{attribute 'linkalways'} 
{attribute 'no_explicit_call' := 'This FB is a CLASS and must be accessed using methods or properties'}
{attribute 'enable_dynamic_creation'}
FUNCTION_BLOCK _ETcVnContoursMatchComparisonMethod EXTENDS EnumDatatypeBase
VAR
	localData : ETcVnContoursMatchComparisonMethod;
	activeData : REFERENCE TO ETcVnContoursMatchComparisonMethod;
	enumBaseDatatype : _DINT(localData);
END_VAR

METHOD PRIVATE AddLocalEnumeration
VAR_INPUT
	Enumeration : T_MAXSTRING;
	Value : ETcVnContoursMatchComparisonMethod;
END_VAR
AddEnumeration(Enumeration, Value);
END_METHOD

PROPERTY PUBLIC Address : PVOID
GET
Address := ADR(activeData);
END_GET
END_PROPERTY

METHOD PUBLIC ClearReference
VAR_INPUT
END_VAR
activeData REF= localData;
SetBaseDatatypeReference();
END_METHOD

METHOD PUBLIC Clone : I_Datatype
VAR
    pClone : POINTER TO _ETcVnContoursMatchComparisonMethod;
END_VAR
pClone := __NEW(_ETcVnContoursMatchComparisonMethod(InitialValue := Value));
Clone := pClone^;
END_METHOD

METHOD FB_init : BOOL
VAR_INPUT
	bInitRetains : BOOL; // if TRUE, the retain variables are initialized (warm start / cold start)
	bInCopyCode : BOOL;  // if TRUE, the instance afterwards gets moved into the copy code (online change)
	InitialValue : ETcVnContoursMatchComparisonMethod;
END_VAR
localData := InitialValue;
AddBaseDatatype(enumBaseDatatype);
ClearReference();

AddLocalEnumeration('TCVN_CMCM_CONTOURS_MATCH_I1', ETcVnContoursMatchComparisonMethod.TCVN_CMCM_CONTOURS_MATCH_I1);
AddLocalEnumeration('TCVN_CMCM_CONTOURS_MATCH_I2', ETcVnContoursMatchComparisonMethod.TCVN_CMCM_CONTOURS_MATCH_I2);
AddLocalEnumeration('TCVN_CMCM_CONTOURS_MATCH_I3', ETcVnContoursMatchComparisonMethod.TCVN_CMCM_CONTOURS_MATCH_I3);
END_METHOD

PROPERTY PUBLIC Identifier : T_MAXSTRING
GET
Identifier := 'ETcVnContoursMatchComparisonMethod';
END_GET
END_PROPERTY

METHOD IsEnumeratorValueEqual : BOOL
VAR_INPUT
	Enumerator : I_KeyValueForwardEnumerator;
END_VAR
VAR
	storedValue : ETcVnContoursMatchComparisonMethod;
END_VAR
IF NOT Enumerator.TryGet(storedValue) THEN
	RETURN;
END_IF

IsEnumeratorValueEqual := storedValue = activeData;
END_METHOD

METHOD PUBLIC MakeReferenceTo
VAR_INPUT
	ReferenceTarget : REFERENCE TO ETcVnContoursMatchComparisonMethod;
END_VAR
activeData REF= ReferenceTarget;
SetBaseDatatypeReference();
END_METHOD

METHOD PROTECTED SetBaseDatatypeReference
VAR_INPUT
END_VAR
enumBaseDatatype.MakeReferenceTo(activeData);
END_METHOD

PROPERTY PUBLIC Size : UDINT
GET
Size := SIZEOF(activeData);
END_GET
END_PROPERTY

METHOD TryMakeReferenceTo : BOOL
VAR_INPUT
	Target : I_Datatype;
END_VAR
VAR
	targetAsEnum : I_EnumDatatype;
	pTargetData : POINTER TO ETcVnContoursMatchComparisonMethod;
END_VAR
IF NOT Target.TryResolveAsEnumDatatype(targetAsEnum) THEN
	RETURN;
END_IF

IF targetAsEnum.Identifier <> Identifier THEN
	RETURN;
END_IF

pTargetData := Target.Address;
activeData REF= pTargetData^;
SetBaseDatatypeReference();
TryMakeReferenceTo := TRUE;
END_METHOD

PROPERTY PUBLIC Value : ETcVnContoursMatchComparisonMethod
GET
Value := activeData;
END_GET
SET
activeData := Value;
END_SET
END_PROPERTY

END_FUNCTION_BLOCK

(* stored: Version 1.1.0.1, ProductVersion 3.1.4024.12
   POU _ETcVnContoursMatchComparisonMethod: Id {6320c7ac-4a20-4d27-9069-a7f3038d260f}, SpecialFunc None
   Folder Constructor: Id {43715b9e-181a-4002-9f04-bbfe65491932}
   Folder Private: Id {24b76ea8-3d87-4bd5-b823-eaf4db1690a0}
   Folder Protected: Id {8dad596b-3852-43a2-9d7f-c0a972f9c5bf}
   Method AddLocalEnumeration: Id {aacbcdb8-417f-406a-8641-65ffb96ca382}
   Property Address: Id {41e68ffc-2ac6-4e42-81cf-445b9953fd0f}
   Get Get: Id {622bf6c0-726c-4f2d-b934-821a43acb118}
   Method ClearReference: Id {6322fd32-6fe5-46ee-a8e2-504fcabac3b0}
   Method Clone: Id {4e0af0c7-82dd-42ab-8102-073387cfe13e}
   Method FB_init: Id {606b60c5-c0aa-483d-b0b3-e0a124ad919b}
   Property Identifier: Id {c3731226-fff0-4380-96ef-611a64cd4edd}
   Get Get: Id {05f77fce-457f-4cdd-8940-3c50851ca9c8}
   Method IsEnumeratorValueEqual: Id {ec134804-4560-4314-921c-f869fcb9d608}
   Method MakeReferenceTo: Id {3cf7d413-75c6-441b-b493-0471d9e9eefa}
   Method SetBaseDatatypeReference: Id {484186ea-a3cf-4827-86cf-cd63758ea302}
   Property Size: Id {9295ed37-4c18-40e6-84ff-42fb8016765c}
   Get Get: Id {0952df95-4b14-45b6-bc77-8703ca96733b}
   Method TryMakeReferenceTo: Id {7474621b-fc45-4290-96a9-b03319fbf558}
   Property Value: Id {f66d77c8-8248-4e1f-bf3a-b7b9c3048d60}
   Get Get: Id {b7acebf9-e05b-4093-98b4-225738c0d782}
   Set Set: Id {20977503-aa10-4023-896d-00acb42d5d65} *)
